FUNCTION_BLOCK fb_cleanIn
VAR_INPUT
	IN: BOOL;
END_VAR
VAR_OUTPUT
END_VAR
VAR
	wait: TON;
	step: INT;
END_VAR

VAR_IN_OUT
	done: BOOL;
END_VAR

CASE step OF
	0:
		IF NOT done THEN
			cleanout.inValve := TRUE;
			wait(IN := TRUE, PT := T#5S);
			step := 1;
		END_IF
	1:
		IF wait.Q THEN
			wait.IN := FALSE;
			cleanout.inValve := FALSE;
			step := 2;
		END_IF
		
	2: 
		step := 0;
		done := TRUE;
	
END_CASE
wait();

END_FUNCTION_BLOCK

(* stored: Version 1.1.0.1, ProductVersion 3.1.4024.5
   POU fb_cleanIn: Id {b2bc3242-131e-4da2-9489-b8575e111113}, SpecialFunc None *)
